{attribute 'qualified_only'}
VAR_GLOBAL
	iInt	: UDINT;
END_VAR

(* stored: Version 1.1.0.1, ProductVersion 3.1.4024.15
   GVL GVL: Id {9748686d-37a2-438d-8b30-65f95070eafd} *)
